FUNCTION INTERNAL _FinalizeEntity : Result
VAR
	i						: UDINT;
END_VAR

IF NOT _Runtime.bInit THEN
	_RegEntity := Err.Init;
	RETURN;
END_IF

IF _Ec.iUnderConstruction = 0 THEN
	_RegEntity := Err.Itf0;
	RETURN;
END_IF

_Ec.iUnderConstruction._IsCompleted := TRUE;

_Ec.nConstructedScopes := _Ec.nConstructedScopes - 1;
IF _Ec.nConstructedScopes > 0 THEN
	FOR i := _Ec.iUnderConstruction.Id TO 1 BY -1 DO
		IF NOT _Ec.iEntity[i]._IsCompleted THEN
			_Ec.iUnderConstruction := _Ec.iEntity[i];
			_FinalizeEntity := Ok;
			RETURN;
		END_IF
	END_FOR
	
	_FinalizeEntity := Err.Udf;
ELSE
	_Ec.iUnderConstruction := 0;
	_FinalizeEntity := Ok;
END_IF

END_FUNCTION

(* stored: Version 1.1.0.1
   POU _FinalizeEntity: Id {82cbd3cc-9cc2-4c0d-b07f-49b218e520bd}, SpecialFunc None *)
